PROGRAM P_Trappe
VAR
	
	
	DigIn3	AT %I* :	BOOL;
	DigIn4	AT %I* :	BOOL;
	DigIn5	AT %I* :	BOOL;
	DigIn6	AT %I* :	BOOL;
	DigIn7	AT %I* :	BOOL;
	DigIn8	AT %I* :	BOOL;
	
	DigOut1 AT %Q*	:	BOOL;
END_VAR

END_PROGRAM

(* stored: Version 1.1.0.1
   POU P_Trappe: Id {83c3eb57-219c-4506-9fd5-12c478d2b64c}, SpecialFunc None *)
